// TIA Portal V20 export
TYPE "LAxisCtrl_typeCamIn"
TITLE = LAxisCtrl_typeCamIn
// Support: tech.team.motioncontrol@siemens.com 
// Fax: +49 (0) 9131/98-1297
   STRUCT
      masterOffset : LReal := 0.0;   // Offset of leading values of cam
      slaveOffset : LReal := 0.0;   // Offset of following values of cam
      masterScaling : LReal := 1.0;   // Scaling the leading values of the cam
      slaveScaling : LReal := 1.0;   // Scaling the following values of the cam
      masterSyncPosition : LReal := 0.0;   // Starting point in the cam/distance from the cam start with reference to the scaled cam
      syncProfileReference : DInt := 1;   // Synchronization profile (0: Synchronization using dynamic parameters; 1: Synchronization using leading value distance; 2: Direct synchronous setting)
      masterStartDistance : LReal := 0.0;   // Leading value distance (when "SyncProfileReference" = 1)
      velocity : LReal := -1.0;   // Velocity for synchronization (when "SyncProfileReference" = 0; Value > 0.0: The specified value is used; Value = 0.0: Not permitted; Value < 0.0: Use of the default value configured in the technology object)
      acceleration : LReal := -1.0;   // Acceleration for synchronization (when "SyncProfileReference" = 0; Value > 0.0: The specified value is used; Value = 0.0: Not permitted; Value < 0.0: Use of the default value configured in the technology object)
      deceleration : LReal := -1.0;   // Deceleration for synchronization (when "SyncProfileReference" = 0; Value > 0.0: The specified value is used; Value = 0.0: Not permitted; Value < 0.0: Use of the default value configured in the technology object)
      jerk : LReal := -1.0;   // Jerk for synchronization (when "SyncProfileReference" = 0; Value > 0.0: Smooth velocity profile, the specified value is used; Value = 0.0: Trapezoid velocity profile; Value < 0.0: Use of the default value configured in the technology object)
      applicationMode : DInt := 0;   // Application of the cam (0: Once/not cyclic; 1: Cyclic ; 2: Cyclic appending)
      syncDirection : DInt := 1;   // Direction for synchronization only in effect for axes with activated modulo setting (1: Forward direction; 2: Backward direction; 3: Shortest way)
   END_STRUCT;
END_TYPE
